(* Logix 5000 project; controller AplicacionAFEbancoDePruebas vendor 1 type 14 code 149 rev 33.12; software revision 33.01 *)

TASK MainTask (continuous, watchdog 500 ms) : MainProgram

MODULES
   Local : vendor 1 type 14 code 149 (Compact 0, rev 33.12)
      Discrete_IO : Embedded (Compact 1, rev 3.1, Output RPI 20 ms)
      PLC : 1769-L32E Ethernet Port (Ethernet 192.168.2.131, rev 20.1)
         PLC_Controller : vendor 1 type 14 code 77 (CompactLogixL32EController 0, rev 20.1, $1600cdba$ RPI 20 ms, $c578c295$ RPI 20 ms, $949708e4$ RPI 20 ms)
      VSD_AFE : vendor 1 type 143 code 8336 (Ethernet 192.168.2.50, rev 6.5, Output RPI 20 ms)
           VSD_AFE:O.LogicCommand_Stop   // Comando de Parada
           VSD_AFE:O.LogicCommand_Start   // Comando de Arranque
          : vendor 1 type 143 code 161 (RhinoBP 10, rev 1.1)
          : vendor 1 type 143 code 416 (RhinoBP 5, rev 1.8)
          : vendor 1 type 143 code 675 (RhinoBP 13, rev 1.1)
          : vendor 1 type 143 code 416 (RhinoBP 4, rev 1.8)
          : vendor 1 type 143 code 4770 (RhinoBP 12, rev 1.1)
          : vendor 1 type 143 code 2724 (RhinoBP 14, rev 1.1)
END_MODULES

TYPE Dinagrama :   // Estructura para el dinagrama
STRUCT
   vPotencia : REAL[500];   // captura del vector de potencia
   vCarga : REAL[500];   // captura del vector de carga
   vPosicion : REAL[500];   // captura del vector posicion
   vProximetro : DINT[500];   // captura del vector del proximetro
   NumeroMuestras : INT;
   enabled : BOOL;
   captura : BOOL;   // Flag que indica la captura del sistema
END_STRUCT
END_TYPE

TYPE LSW :   // Drive - Logic Status Word
STRUCT
   Faulted : BOOL;
   Warning : BOOL;
   RunForward : BOOL;
   RunReverse : BOOL;
   Ready : BOOL;
   RemoteRef : BOOL;
   RemoteCrtl : BOOL;
   AtSpeed : BOOL;
END_STRUCT
END_TYPE

TYPE SWC :
STRUCT
   Dinagrama : Dinagrama;
   VSD : VSD;
   entradasDigitales : INT;   // Entradas Digitales
   salidasDigitales : INT;   // Salidas Digitales
   entradasAnalogas : REAL[4];   // Entradas Analogas del PLC
   salidasAnalogas : REAL[4];
END_STRUCT
END_TYPE

TYPE VSD :   // VSD
STRUCT
   VSD_O : AB:PowerFlex755T_E_31635488:O:0;
   VSD_I : AB:PowerFlex755T_E_2B0A69C5:I:0;
END_STRUCT
END_TYPE

VAR_GLOBAL   (* controller tags *)
   SRP_Displacement_Actual : REAL := 76.0;   // Variable de Simulacion PLC DC de Desplazamiento
   SRP_Load_Actual : REAL;   // Variable de simulacion PLC DC de Carga
   SRP_SimActualStroke : DINT;   // Variable Simulación de PLC Variador DC
   SWC : SWC := (Dinagrama.vPotencia[1] := 0.009212976, Dinagrama.vPotencia[2] := 0.009230624, Dinagrama.vPotencia[3] := 0.015417241, Dinagrama.vPotencia[4] := 0.008623187, Dinagrama.vPotencia[5] := 0.008543681, Dinagrama.vPotencia[8] := 0.008029409, Dinagrama.vPotencia[9] := 0.00787571, Dinagrama.vPotencia[10] := 0.007877604, Dinagrama.vPotencia[11] := 0.0076953056, Dinagrama.vPotencia[17] := 0.0067351083, Dinagrama.vPotencia[18] := 0.0063158795, Dinagrama.vPotencia[20] := 0.0061844666, Dinagrama.vPotencia[27] := 0.005079035, Dinagrama.vPotencia[31] := 0.004283302, Dinagrama.vPotencia[40] := 0.00299628, Dinagrama.vPotencia[41] := 0.002841949, Dinagrama.vPotencia[44] := 0.0020909396, Dinagrama.vPotencia[45] := 0.0019782658, Dinagrama.vPotencia[48] := 0.0015723343, Dinagrama.vPotencia[50] := 0.0012871687, Dinagrama.vPotencia[51] := 0.0010955968, Dinagrama.vPotencia[52] := 0.0009932568, Dinagrama.vPotencia[122] := 0.0128360065, Dinagrama.vPotencia[123] := 0.012979752, Dinagrama.vPotencia[126] := 0.013105653, Dinagrama.vPotencia[127] := 0.012908061, Dinagrama.vPotencia[129] := 0.013102764, Dinagrama.vPotencia[130] := 0.012823998, Dinagrama.vPotencia[133] := 0.012842169, Dinagrama.vPotencia[134] := 0.013001867, Dinagrama.vPotencia[135] := 0.012793231, Dinagrama.vPotencia[137] := 0.01302348, Dinagrama.vPotencia[139] := 0.012982651, Dinagrama.vPotencia[140] := 0.013010237, Dinagrama.vPotencia[141] := 0.0128319105, Dinagrama.vPotencia[143] := 0.01302347, Dinagrama.vPotencia[147] := 0.012924826, Dinagrama.vPotencia[150] := 0.0130830435, Dinagrama.vPotencia[151] := 0.013074962, Dinagrama.vPotencia[152] := 0.012869947, Dinagrama.vPotencia[154] := 0.013073334, Dinagrama.vPotencia[157] := 0.012900667, Dinagrama.vPotencia[158] := 0.013004556, Dinagrama.vPotencia[160] := 0.012767854, Dinagrama.vPotencia[161] := 0.013025847, Dinagrama.vPotencia[162] := 0.0129110655, Dinagrama.vPotencia[164] := 0.012972139, Dinagrama.vPotencia[165] := 0.0128591545, Dinagrama.vPotencia[168] := 0.012745578, Dinagrama.vPotencia[170] := 0.012901854, Dinagrama.vPotencia[171] := 0.01275341, Dinagrama.vPotencia[174] := 0.012726286, Dinagrama.vPotencia[175] := 0.012993207, Dinagrama.vPotencia[178] := 0.0130504845, Dinagrama.vPotencia[180] := 0.012934142, Dinagrama.vPotencia[182] := 0.025404012, Dinagrama.vPotencia[185] := 0.01278092, Dinagrama.vPotencia[189] := 0.013054937, Dinagrama.vPotencia[193] := 0.012787204, Dinagrama.vPotencia[196] := 0.012795925,
        Dinagrama.vPotencia[198] := 0.012868085, Dinagrama.vPotencia[199] := 0.013061226, Dinagrama.vPotencia[201] := 0.01286367, Dinagrama.vPotencia[203] := 0.026164604, Dinagrama.vPotencia[206] := 0.012775595, Dinagrama.vPotencia[208] := 0.013000788, Dinagrama.vPotencia[216] := 0.013077236, Dinagrama.vPotencia[227] := 0.013020926, Dinagrama.vPotencia[230] := 0.012999376, Dinagrama.vPotencia[234] := 0.0128271105, Dinagrama.vPotencia[235] := 0.0131178405, Dinagrama.vPotencia[241] := 0.012931585, Dinagrama.vPotencia[242] := 0.012805867, Dinagrama.vPotencia[244] := 0.025965039, Dinagrama.vPotencia[246] := 0.012987479, Dinagrama.vCarga[1] := 1.0, Dinagrama.vCarga[2] := 1.0, Dinagrama.vCarga[3] := 2.0, Dinagrama.vCarga[4] := 2.0, Dinagrama.vCarga[5] := 3.0, Dinagrama.vCarga[6] := 3.0, Dinagrama.vCarga[7] := 4.0, Dinagrama.vCarga[8] := 4.0, Dinagrama.vCarga[9] := 5.0, Dinagrama.vCarga[10] := 6.0, Dinagrama.vCarga[11] := 6.0, Dinagrama.vCarga[12] := 7.0, Dinagrama.vCarga[13] := 8.0, Dinagrama.vCarga[14] := 8.0, Dinagrama.vCarga[15] := 9.0, Dinagrama.vCarga[16] := 9.0, Dinagrama.vCarga[17] := 10.0, Dinagrama.vCarga[18] := 10.0, Dinagrama.vCarga[19] := 11.0, Dinagrama.vCarga[20] := 12.0, Dinagrama.vCarga[21] := 12.0, Dinagrama.vCarga[22] := 13.0, Dinagrama.vCarga[23] := 13.0, Dinagrama.vCarga[24] := 14.0, Dinagrama.vCarga[25] := 14.0, Dinagrama.vCarga[26] := 15.0, Dinagrama.vCarga[27] := 15.0, Dinagrama.vCarga[28] := 16.0, Dinagrama.vCarga[29] := 17.0, Dinagrama.vCarga[30] := 17.0, Dinagrama.vCarga[31] := 18.0, Dinagrama.vCarga[32] := 19.0, Dinagrama.vCarga[33] := 19.0, Dinagrama.vCarga[34] := 19.0, Dinagrama.vCarga[35] := 20.0, Dinagrama.vCarga[36] := 21.0, Dinagrama.vCarga[37] := 21.0, Dinagrama.vCarga[38] := 22.0, Dinagrama.vCarga[39] := 22.0, Dinagrama.vCarga[40] := 23.0, Dinagrama.vCarga[41] := 24.0, Dinagrama.vCarga[42] := 24.0, Dinagrama.vCarga[43] := 25.0, Dinagrama.vCarga[44] := 25.0, Dinagrama.vCarga[45] := 26.0,
        Dinagrama.vCarga[46] := 26.0, Dinagrama.vCarga[47] := 27.0, Dinagrama.vCarga[48] := 28.0, Dinagrama.vCarga[49] := 28.0, Dinagrama.vCarga[50] := 29.0, Dinagrama.vCarga[51] := 29.0, Dinagrama.vCarga[52] := 30.0, Dinagrama.vCarga[53] := 30.0, Dinagrama.vCarga[54] := 31.0, Dinagrama.vCarga[55] := 31.0, Dinagrama.vCarga[56] := 32.0, Dinagrama.vCarga[57] := 33.0, Dinagrama.vCarga[58] := 33.0, Dinagrama.vCarga[59] := 34.0, Dinagrama.vCarga[60] := 34.0, Dinagrama.vCarga[61] := 35.0, Dinagrama.vCarga[62] := 35.0, Dinagrama.vCarga[63] := 36.0, Dinagrama.vCarga[64] := 37.0, Dinagrama.vCarga[65] := 37.0, Dinagrama.vCarga[66] := 38.0, Dinagrama.vCarga[67] := 38.0, Dinagrama.vCarga[68] := 39.0, Dinagrama.vCarga[69] := 40.0, Dinagrama.vCarga[70] := 40.0, Dinagrama.vCarga[71] := 41.0, Dinagrama.vCarga[72] := 41.0, Dinagrama.vCarga[73] := 42.0, Dinagrama.vCarga[74] := 42.0, Dinagrama.vCarga[75] := 43.0, Dinagrama.vCarga[76] := 43.0, Dinagrama.vCarga[77] := 44.0, Dinagrama.vCarga[78] := 45.0, Dinagrama.vCarga[79] := 45.0, Dinagrama.vCarga[80] := 46.0, Dinagrama.vCarga[81] := 46.0, Dinagrama.vCarga[82] := 47.0, Dinagrama.vCarga[83] := 47.0, Dinagrama.vCarga[84] := 48.0, Dinagrama.vCarga[85] := 49.0, Dinagrama.vCarga[86] := 49.0, Dinagrama.vCarga[87] := 50.0, Dinagrama.vCarga[88] := 50.0, Dinagrama.vCarga[89] := 51.0, Dinagrama.vCarga[90] := 52.0, Dinagrama.vCarga[91] := 52.0, Dinagrama.vCarga[92] := 53.0, Dinagrama.vCarga[93] := 53.0, Dinagrama.vCarga[94] := 54.0, Dinagrama.vCarga[95] := 54.0, Dinagrama.vCarga[96] := 55.0, Dinagrama.vCarga[97] := 56.0, Dinagrama.vCarga[98] := 56.0, Dinagrama.vCarga[99] := 57.0, Dinagrama.vCarga[100] := 57.0, Dinagrama.vCarga[101] := 58.0, Dinagrama.vCarga[102] := 58.0, Dinagrama.vCarga[103] := 59.0, Dinagrama.vCarga[104] := 59.0, Dinagrama.vCarga[105] := 60.0,
        Dinagrama.vCarga[106] := 61.0, Dinagrama.vCarga[107] := 61.0, Dinagrama.vCarga[108] := 62.0, Dinagrama.vCarga[109] := 63.0, Dinagrama.vCarga[110] := 63.0, Dinagrama.vCarga[111] := 64.0, Dinagrama.vCarga[112] := 64.0, Dinagrama.vCarga[113] := 65.0, Dinagrama.vCarga[114] := 65.0, Dinagrama.vCarga[115] := 66.0, Dinagrama.vCarga[116] := 66.0, Dinagrama.vCarga[117] := 67.0, Dinagrama.vCarga[118] := 68.0, Dinagrama.vCarga[119] := 68.0, Dinagrama.vCarga[120] := 68.0, Dinagrama.vCarga[121] := 69.0, Dinagrama.vCarga[122] := 70.0, Dinagrama.vCarga[123] := 71.0, Dinagrama.vCarga[124] := 71.0, Dinagrama.vCarga[125] := 72.0, Dinagrama.vCarga[126] := 72.0, Dinagrama.vCarga[127] := 73.0, Dinagrama.vCarga[128] := 74.0, Dinagrama.vCarga[129] := 74.0, Dinagrama.vCarga[130] := 74.0, Dinagrama.vCarga[131] := 75.0, Dinagrama.vCarga[132] := 76.0, Dinagrama.vCarga[133] := 76.0, Dinagrama.vCarga[134] := 77.0, Dinagrama.vCarga[135] := 78.0, Dinagrama.vCarga[136] := 78.0, Dinagrama.vCarga[137] := 79.0, Dinagrama.vCarga[138] := 79.0, Dinagrama.vCarga[139] := 80.0, Dinagrama.vCarga[140] := 80.0, Dinagrama.vCarga[141] := 81.0, Dinagrama.vCarga[142] := 81.0, Dinagrama.vCarga[143] := 82.0, Dinagrama.vCarga[144] := 83.0, Dinagrama.vCarga[145] := 83.0, Dinagrama.vCarga[146] := 84.0, Dinagrama.vCarga[147] := 84.0, Dinagrama.vCarga[148] := 85.0, Dinagrama.vCarga[149] := 85.0, Dinagrama.vCarga[150] := 86.0, Dinagrama.vCarga[151] := 87.0, Dinagrama.vCarga[152] := 87.0, Dinagrama.vCarga[153] := 88.0, Dinagrama.vCarga[154] := 88.0, Dinagrama.vCarga[155] := 89.0, Dinagrama.vCarga[156] := 90.0, Dinagrama.vCarga[157] := 90.0, Dinagrama.vCarga[158] := 90.0, Dinagrama.vCarga[159] := 91.0, Dinagrama.vCarga[160] := 92.0, Dinagrama.vCarga[161] := 92.0, Dinagrama.vCarga[162] := 93.0, Dinagrama.vCarga[163] := 93.0, Dinagrama.vCarga[164] := 94.0, Dinagrama.vCarga[165] := 94.0,
        Dinagrama.vCarga[166] := 95.0, Dinagrama.vCarga[167] := 96.0, Dinagrama.vCarga[168] := 96.0, Dinagrama.vCarga[169] := 97.0, Dinagrama.vCarga[170] := 97.0, Dinagrama.vCarga[171] := 98.0, Dinagrama.vCarga[172] := 99.0, Dinagrama.vCarga[173] := 99.0, Dinagrama.vCarga[174] := 100.0, Dinagrama.vCarga[175] := 100.0, Dinagrama.vCarga[176] := 101.0, Dinagrama.vCarga[177] := 101.0, Dinagrama.vCarga[178] := 102.0, Dinagrama.vCarga[179] := 103.0, Dinagrama.vCarga[180] := 103.0, Dinagrama.vCarga[181] := 104.0, Dinagrama.vCarga[182] := 104.0, Dinagrama.vCarga[183] := 105.0, Dinagrama.vCarga[184] := 106.0, Dinagrama.vCarga[185] := 106.0, Dinagrama.vCarga[186] := 107.0, Dinagrama.vCarga[187] := 107.0, Dinagrama.vCarga[188] := 108.0, Dinagrama.vCarga[189] := 108.0, Dinagrama.vCarga[190] := 109.0, Dinagrama.vCarga[191] := 109.0, Dinagrama.vCarga[192] := 110.0, Dinagrama.vCarga[193] := 111.0, Dinagrama.vCarga[194] := 111.0, Dinagrama.vCarga[195] := 112.0, Dinagrama.vCarga[196] := 112.0, Dinagrama.vCarga[197] := 113.0, Dinagrama.vCarga[198] := 113.0, Dinagrama.vCarga[199] := 114.0, Dinagrama.vCarga[200] := 115.0, Dinagrama.vCarga[201] := 115.0, Dinagrama.vCarga[202] := 116.0, Dinagrama.vCarga[203] := 116.0, Dinagrama.vCarga[204] := 117.0, Dinagrama.vCarga[205] := 118.0, Dinagrama.vCarga[206] := 118.0, Dinagrama.vCarga[207] := 118.0, Dinagrama.vCarga[208] := 119.0, Dinagrama.vCarga[209] := 120.0, Dinagrama.vCarga[210] := 120.0, Dinagrama.vCarga[211] := 121.0, Dinagrama.vCarga[212] := 121.0, Dinagrama.vCarga[213] := 122.0, Dinagrama.vCarga[214] := 123.0, Dinagrama.vCarga[215] := 123.0, Dinagrama.vCarga[216] := 124.0, Dinagrama.vCarga[217] := 124.0, Dinagrama.vCarga[218] := 125.0, Dinagrama.vCarga[219] := 125.0, Dinagrama.vCarga[220] := 126.0, Dinagrama.vCarga[221] := 127.0, Dinagrama.vCarga[222] := 127.0, Dinagrama.vCarga[223] := 128.0, Dinagrama.vCarga[224] := 128.0, Dinagrama.vCarga[225] := 129.0,
        Dinagrama.vCarga[226] := 129.0, Dinagrama.vCarga[227] := 130.0, Dinagrama.vCarga[228] := 130.0, Dinagrama.vCarga[229] := 131.0, Dinagrama.vCarga[230] := 132.0, Dinagrama.vCarga[231] := 132.0, Dinagrama.vCarga[232] := 133.0, Dinagrama.vCarga[233] := 134.0, Dinagrama.vCarga[234] := 134.0, Dinagrama.vCarga[235] := 134.0, Dinagrama.vCarga[236] := 135.0, Dinagrama.vCarga[237] := 136.0, Dinagrama.vCarga[238] := 136.0, Dinagrama.vCarga[239] := 137.0, Dinagrama.vCarga[240] := 137.0, Dinagrama.vCarga[241] := 138.0, Dinagrama.vCarga[242] := 139.0, Dinagrama.vCarga[243] := 139.0, Dinagrama.vCarga[244] := 140.0, Dinagrama.vCarga[245] := 140.0, Dinagrama.vCarga[246] := 140.0, Dinagrama.vCarga[247] := 140.0, Dinagrama.vPosicion[1] := 12.0, Dinagrama.vPosicion[2] := 12.0, Dinagrama.vPosicion[3] := 5.0, Dinagrama.vPosicion[4] := 5.0, Dinagrama.vPosicion[5] := 6.0, Dinagrama.vPosicion[6] := 6.0, Dinagrama.vPosicion[7] := 7.0, Dinagrama.vPosicion[8] := 89.0, Dinagrama.vPosicion[9] := 89.0, Dinagrama.vPosicion[10] := 9.0, Dinagrama.vPosicion[11] := 9.0, Dinagrama.vPosicion[12] := 3.0, Dinagrama.vPosicion[13] := 4.0, Dinagrama.vPosicion[14] := 4.0, Dinagrama.vPosicion[15] := 6.0, Dinagrama.vPosicion[16] := 6.0, Dinagrama.vPosicion[20] := 8.0, Dinagrama.vPosicion[21] := 8.0, Dinagrama.vPosicion[24] := 56.0, Dinagrama.vPosicion[25] := 56.0, Dinagrama.vPosicion[28] := 56.0, Dinagrama.vPosicion[31] := 56.0, Dinagrama.vPosicion[36] := 8765.0, Dinagrama.vPosicion[37] := 8765.0, Dinagrama.vPosicion[41] := 5678.0, Dinagrama.vPosicion[42] := 5678.0, Dinagrama.vPosicion[45] := 5678.0, Dinagrama.vPosicion[46] := 5678.0, Dinagrama.vPosicion[47] := 567.0, Dinagrama.vPosicion[48] := 8.0, Dinagrama.vPosicion[49] := 8.0, Dinagrama.vPosicion[50] := 324.0, Dinagrama.vPosicion[51] := 324.0, Dinagrama.vPosicion[54] := 234.0, Dinagrama.vPosicion[55] := 234.0, Dinagrama.vPosicion[56] := 324.0, Dinagrama.vPosicion[57] := 234.0, Dinagrama.vPosicion[58] := 234.0,
        Dinagrama.vPosicion[59] := 234.0, Dinagrama.vPosicion[60] := 234.0, Dinagrama.vPosicion[61] := 342.0, Dinagrama.vPosicion[62] := 342.0, Dinagrama.vPosicion[63] := 34.0, Dinagrama.vPosicion[75] := 432.0, Dinagrama.vPosicion[76] := 432.0, Dinagrama.vPosicion[78] := 4.0, Dinagrama.vPosicion[79] := 4.0, Dinagrama.vPosicion[80] := 4.0, Dinagrama.vPosicion[81] := 4.0, Dinagrama.vPosicion[82] := 4.0, Dinagrama.vPosicion[83] := 4.0, Dinagrama.vPosicion[84] := 4.0, Dinagrama.vPosicion[87] := 3.0, Dinagrama.vPosicion[88] := 3.0, Dinagrama.vPosicion[90] := 2.0, Dinagrama.vPosicion[91] := 2.0, Dinagrama.vPosicion[96] := 245.0, Dinagrama.vPosicion[97] := 2345.0, Dinagrama.vPosicion[98] := 2345.0, Dinagrama.vPosicion[99] := 2345.0, Dinagrama.vPosicion[100] := 2345.0, Dinagrama.vPosicion[101] := 724.0, Dinagrama.vPosicion[102] := 724.0, Dinagrama.vPosicion[103] := 4325.0, Dinagrama.vPosicion[104] := 4325.0, Dinagrama.vPosicion[105] := 3245.0, Dinagrama.vPosicion[106] := 2345.0, Dinagrama.vPosicion[107] := 2345.0, Dinagrama.vPosicion[150] := 2345.0, Dinagrama.vPosicion[155] := 2345.0, Dinagrama.vPosicion[159] := 2345.0, Dinagrama.vPosicion[160] := 2345.0, Dinagrama.vPosicion[161] := 2345.0, Dinagrama.vPosicion[171] := 234.0, Dinagrama.vPosicion[172] := 4.0, Dinagrama.vPosicion[173] := 4.0, Dinagrama.vPosicion[174] := 2.0, Dinagrama.vPosicion[175] := 2.0, Dinagrama.vPosicion[176] := 3.0, Dinagrama.vPosicion[177] := 3.0, Dinagrama.vPosicion[178] := 45.0, Dinagrama.vPosicion[179] := 2345.0, Dinagrama.vPosicion[180] := 2345.0, Dinagrama.vPosicion[181] := 2345.0, Dinagrama.vPosicion[182] := 2345.0, Dinagrama.vPosicion[183] := 5234.0, Dinagrama.vPosicion[184] := 354.0, Dinagrama.vPosicion[185] := 354.0, Dinagrama.vProximetro[0] := 1, Dinagrama.vProximetro[1] := 1, Dinagrama.vProximetro[2] := 1, Dinagrama.vProximetro[3] := 1, Dinagrama.vProximetro[4] := 1, Dinagrama.vProximetro[5] := 1, Dinagrama.vProximetro[6] := 1, Dinagrama.vProximetro[7] := 1, Dinagrama.vProximetro[8] := 1, Dinagrama.vProximetro[9] := 1,
        Dinagrama.vProximetro[10] := 1, Dinagrama.vProximetro[11] := 1, Dinagrama.vProximetro[246] := 1, Dinagrama.vProximetro[248] := 1, Dinagrama.vProximetro[249] := 1, Dinagrama.vProximetro[250] := 1, Dinagrama.vProximetro[251] := 1, Dinagrama.vProximetro[252] := 1, Dinagrama.vProximetro[253] := 1, Dinagrama.vProximetro[254] := 1, Dinagrama.vProximetro[255] := 1, Dinagrama.vProximetro[256] := 1, Dinagrama.vProximetro[257] := 1, Dinagrama.vProximetro[258] := 1, Dinagrama.vProximetro[494] := 1, Dinagrama.vProximetro[495] := 1, Dinagrama.vProximetro[496] := 1, Dinagrama.vProximetro[497] := 1, Dinagrama.vProximetro[498] := 1, Dinagrama.vProximetro[499] := 1, Dinagrama.NumeroMuestras := 120, VSD.VSD_O.P10_VRefAStpt := 6.3158, VSD.VSD_I.DriveStatus := 2#1010_0001_0000_0000_0000_0100_0000_1101, VSD.VSD_I.DriveStatus_Ready := 1, VSD.VSD_I.DriveStatus_CommandDir := 1, VSD.VSD_I.DriveStatus_ActualDir := 1, VSD.VSD_I.DriveStatus_SpdRefBit0 := 1, VSD.VSD_I.DriveStatus_AtZeroSpeed := 1, VSD.VSD_I.DriveStatus_EnableOn := 1, VSD.VSD_I.DriveStatus_Regen := 1, VSD.VSD_I.P10_VRefCommanded := 6.3158, VSD.VSD_I.DCBusVolts := 704.1641, VSD.VSD_I.P10_HeatsnkTemp := 20.0, VSD.VSD_I.ElapsedRunTime := 18.422, VSD.VSD_I.LastFaultCode := 14126, VSD.VSD_I.ElapsedkWH := -9591, entradasDigitales := 3, entradasAnalogas[0] := -1.7e-44, entradasAnalogas[1] := -9.176336e+29, entradasAnalogas[2] := 3.8693e-41, entradasAnalogas[3] := 6.66079e-40, salidasAnalogas[0] := 1.e-45, salidasAnalogas[1] := 6.e-45, salidasAnalogas[2] := 4.e-45);
        .Dinagrama.enabled   // Habilitar Adquision
END_VAR

PROGRAM MainProgram   (* main routine R000_MainRoutine *)
VAR
   Captura : BOOL;
   contadorAux : ALIAS FOR counter[0].ACC;
   counter : COUNTER[10];
   Enabled : BOOL;
   Flag : BOOL;
   habilitar : DINT;
   myoneshot : BOOL[32];
        [0]   // oneshot toogle bot dinagrama
        [1]   // oneshor reset del ocntador
        [2]   // reset de la flag cuando se habilita y se deshabilita
   Proximetro_Virtual : ALIAS FOR SRP_SimActualStroke;
   SPM_Reference : REAL := 8.5;
   timer : TIMER[10] := ([0].PRE := 29);
        [0]   // Tiempo Muestreo
END_VAR

ROUTINE R000_MainRoutine   (* ladder *)
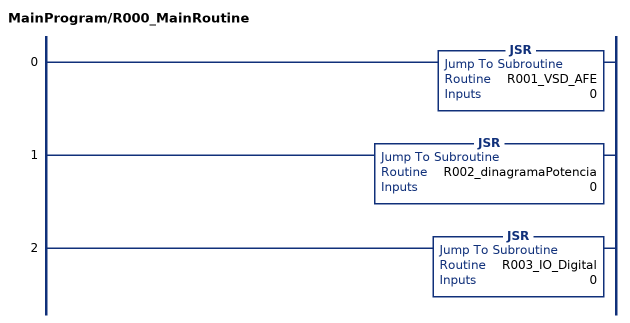
   0: JSR(R001_VSD_AFE,0);
   1: JSR(R002_dinagramaPotencia,0);
   2: JSR(R003_IO_Digital,0);
END_ROUTINE

ROUTINE R001_VSD_AFE   (* ladder *)
// Comandos Basicos de Operación de VSD AFE
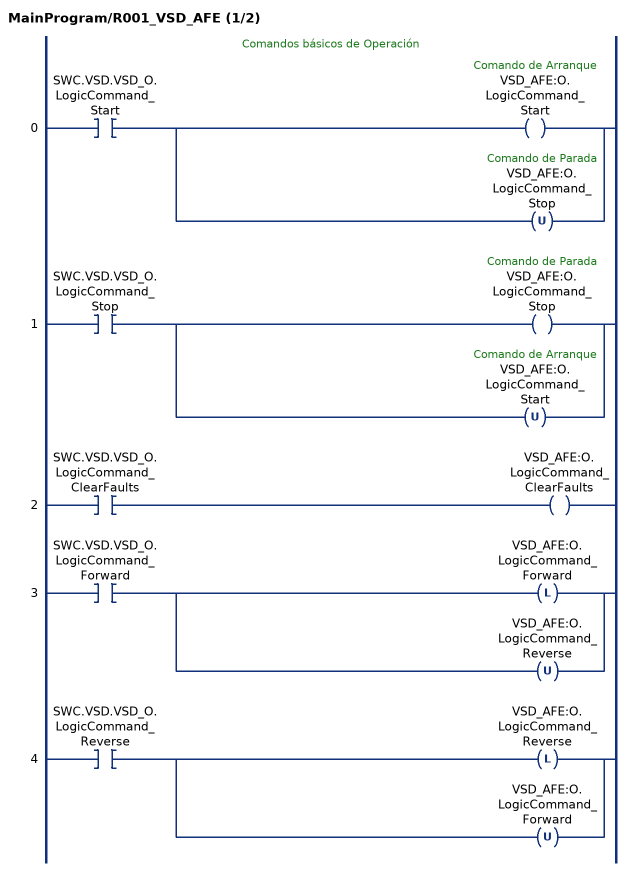
   // Comandos básicos de Operación
   0: XIC(SWC.VSD.VSD_O.LogicCommand_Start)[OTE(VSD_AFE:O.LogicCommand_Start) ,OTU(VSD_AFE:O.LogicCommand_Stop) ];
   1: XIC(SWC.VSD.VSD_O.LogicCommand_Stop)[OTE(VSD_AFE:O.LogicCommand_Stop) ,OTU(VSD_AFE:O.LogicCommand_Start) ];
   2: XIC(SWC.VSD.VSD_O.LogicCommand_ClearFaults)OTE(VSD_AFE:O.LogicCommand_ClearFaults);
   3: XIC(SWC.VSD.VSD_O.LogicCommand_Forward)[OTL(VSD_AFE:O.LogicCommand_Forward) ,OTU(VSD_AFE:O.LogicCommand_Reverse) ];
   4: XIC(SWC.VSD.VSD_O.LogicCommand_Reverse)[OTL(VSD_AFE:O.LogicCommand_Reverse) ,OTU(VSD_AFE:O.LogicCommand_Forward) ];
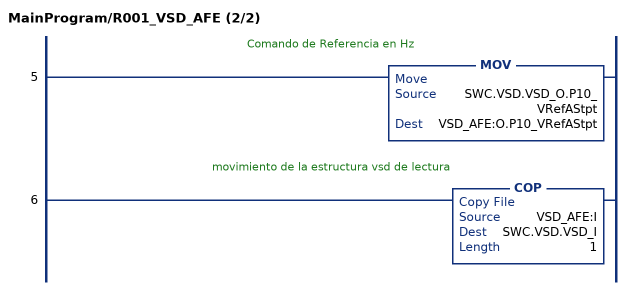
   // Comando de Referencia en Hz
   5: MOV(SWC.VSD.VSD_O.P10_VRefAStpt,VSD_AFE:O.P10_VRefAStpt);
   // movimiento de la estructura vsd de lectura
   6: COP(VSD_AFE:I,SWC.VSD.VSD_I,1);
END_ROUTINE

ROUTINE R002_dinagramaPotencia   (* ladder *)
// Adquisión de los diferentes strokes para la captura del dinagrama de superficie
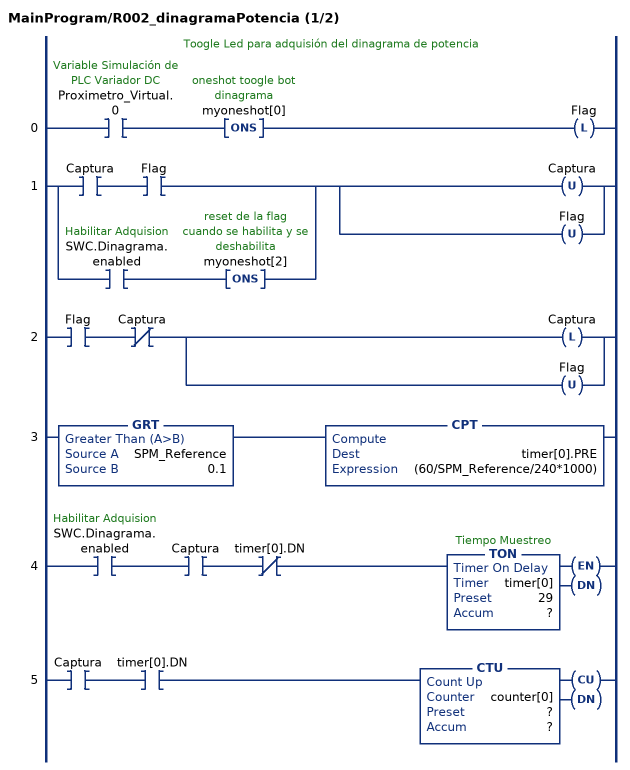
   // Toogle Led para adquisión del dinagrama de potencia
   0: XIC(Proximetro_Virtual.0)ONS(myoneshot[0])OTL(Flag);
   1: [XIC(Captura) XIC(Flag) ,XIC(SWC.Dinagrama.enabled) ONS(myoneshot[2]) ][OTU(Captura) ,OTU(Flag) ];
   2: XIC(Flag)XIO(Captura)[OTL(Captura) ,OTU(Flag) ];
   3: GRT(SPM_Reference,0.1)CPT(timer[0].PRE,(60/SPM_Reference/240*1000));
   4: XIC(SWC.Dinagrama.enabled)XIC(Captura)XIO(timer[0].DN)TON(timer[0],?,?);
   5: XIC(Captura)XIC(timer[0].DN)CTU(counter[0],?,?);
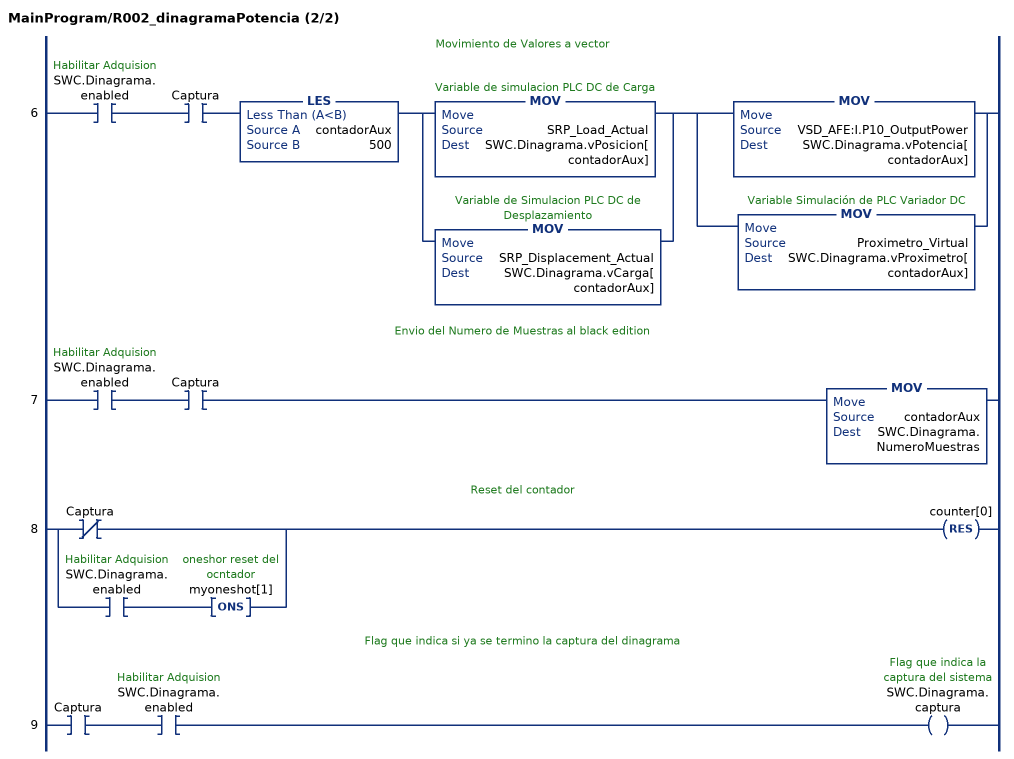
   // Movimiento de Valores a vector
   6: XIC(SWC.Dinagrama.enabled)XIC(Captura)LES(contadorAux,500)[MOV(SRP_Load_Actual,SWC.Dinagrama.vPosicion[contadorAux]) ,MOV(SRP_Displacement_Actual,SWC.Dinagrama.vCarga[contadorAux]) ][MOV(VSD_AFE:I.P10_OutputPower,SWC.Dinagrama.vPotencia[contadorAux]) ,MOV(Proximetro_Virtual,SWC.Dinagrama.vProximetro[contadorAux]) ];
   // Envio del Numero de Muestras al black edition
   7: XIC(SWC.Dinagrama.enabled)XIC(Captura)MOV(contadorAux,SWC.Dinagrama.NumeroMuestras);
   // Reset del contador
   8: [XIO(Captura) ,XIC(SWC.Dinagrama.enabled) ONS(myoneshot[1]) ]RES(counter[0]);
   // Flag que indica si ya se termino la captura del dinagrama
   9: XIC(Captura)XIC(SWC.Dinagrama.enabled)OTE(SWC.Dinagrama.captura);
END_ROUTINE

ROUTINE R003_IO_Digital   (* ladder *)
// Entradas Digitales
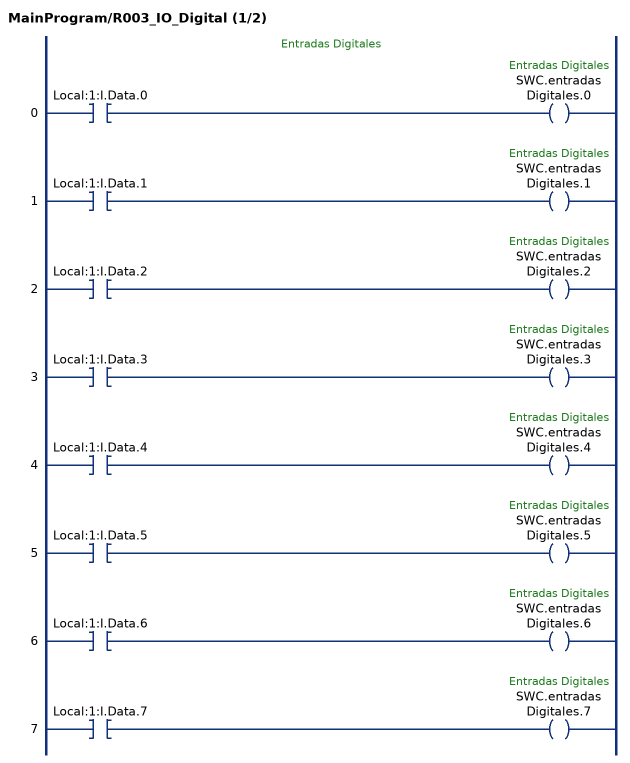
   // Entradas Digitales
   0: XIC(Local:1:I.Data.0)OTE(SWC.entradasDigitales.0);
   1: XIC(Local:1:I.Data.1)OTE(SWC.entradasDigitales.1);
   2: XIC(Local:1:I.Data.2)OTE(SWC.entradasDigitales.2);
   3: XIC(Local:1:I.Data.3)OTE(SWC.entradasDigitales.3);
   4: XIC(Local:1:I.Data.4)OTE(SWC.entradasDigitales.4);
   5: XIC(Local:1:I.Data.5)OTE(SWC.entradasDigitales.5);
   6: XIC(Local:1:I.Data.6)OTE(SWC.entradasDigitales.6);
   7: XIC(Local:1:I.Data.7)OTE(SWC.entradasDigitales.7);
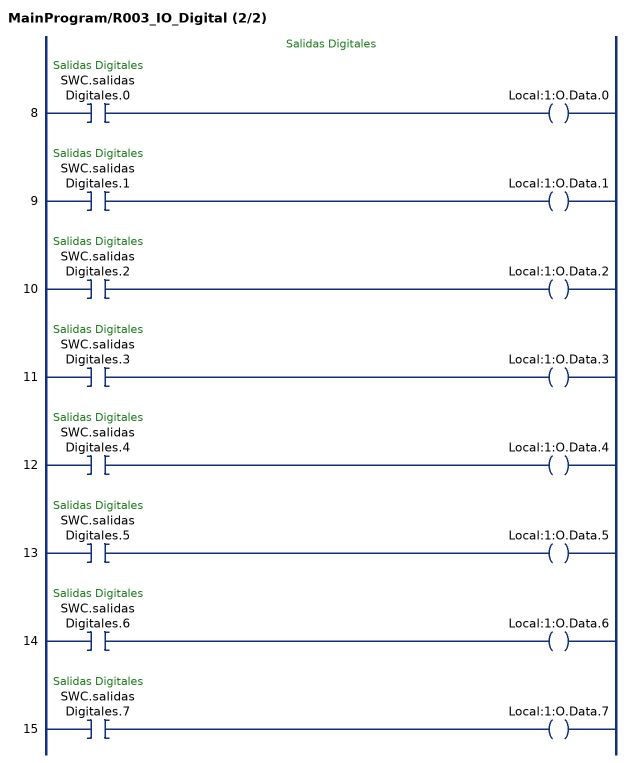
   // Salidas Digitales
   8: XIC(SWC.salidasDigitales.0)OTE(Local:1:O.Data.0);
   9: XIC(SWC.salidasDigitales.1)OTE(Local:1:O.Data.1);
   10: XIC(SWC.salidasDigitales.2)OTE(Local:1:O.Data.2);
   11: XIC(SWC.salidasDigitales.3)OTE(Local:1:O.Data.3);
   12: XIC(SWC.salidasDigitales.4)OTE(Local:1:O.Data.4);
   13: XIC(SWC.salidasDigitales.5)OTE(Local:1:O.Data.5);
   14: XIC(SWC.salidasDigitales.6)OTE(Local:1:O.Data.6);
   15: XIC(SWC.salidasDigitales.7)OTE(Local:1:O.Data.7);
END_ROUTINE
END_PROGRAM
